{attribute 'qualified_only'}
{attribute 'strict'}
TYPE SortOrder :
(
	Ascending,
	Descending
);
END_TYPE

(* stored: Version 1.1.0.1
   EnumerationTextList SortOrder: Id {00d7a571-b6f2-0d82-23f6-8206b5c22cc7} *)
